ABB RAPID module: Module1.mod

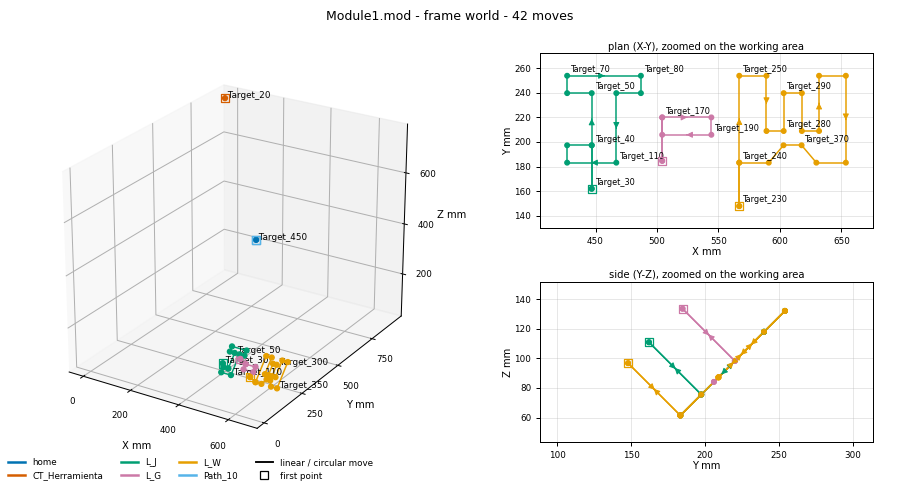
[picture p0: tool path of Module1.mod in frame world, 42 of 42 moves have a stored position in this frame; points joined in program order, loops and branches not executed]
MODULE Module1
    CONST robtarget Target_10:=[[-222.343363548,254.362,580.474563215],[0.5,-0.707106782,0.5,0],[0,-2,1,0],[9E+09,9E+09,9E+09,9E+09,9E+09,9E+09]];
    CONST robtarget Target_20:=[[-918.327354836,-454.935,-37.497165761],[0,0.923879533,0,-0.382683432],[0,0,0,0],[9E+09,9E+09,9E+09,9E+09,9E+09,9E+09]];
    CONST robtarget Target_30:=[[80.000242707,20.000268516,50.000191823],[0,0.707106778,0.707106785,0],[0,0,0,0],[9E+09,9E+09,9E+09,9E+09,9E+09,9E+09]];
    CONST robtarget Target_40:=[[80.000242721,20.000268516,0.000191823],[0,0.707106778,0.707106785,0],[0,0,0,0],[9E+09,9E+09,9E+09,9E+09,9E+09,9E+09]];
    CONST robtarget Target_50:=[[20.000242721,20.000268516,0.000191806],[0,0.707106778,0.707106785,0],[0,0,0,0],[9E+09,9E+09,9E+09,9E+09,9E+09,9E+09]];
    CONST robtarget Target_60:=[[20.000242721,0.000268516,0.000191806],[0,0.707106778,0.707106785,0],[0,0,0,0],[9E+09,9E+09,9E+09,9E+09,9E+09,9E+09]];
    CONST robtarget Target_70:=[[0.000242721,0.000268516,0.000191801],[0,0.707106778,0.707106785,0],[0,0,0,0],[9E+09,9E+09,9E+09,9E+09,9E+09,9E+09]];
    CONST robtarget Target_80:=[[0.000242721,60.000268516,0.000191801],[0,0.707106778,0.707106785,0],[0,0,0,0],[9E+09,9E+09,9E+09,9E+09,9E+09,9E+09]];
    CONST robtarget Target_90:=[[20.000242721,60.000268516,0.000191806],[0,0.707106778,0.707106785,0],[0,0,0,0],[9E+09,9E+09,9E+09,9E+09,9E+09,9E+09]];
    CONST robtarget Target_100:=[[20.000242721,40.000268516,0.000191806],[0,0.707106778,0.707106785,0],[0,0,0,0],[9E+09,9E+09,9E+09,9E+09,9E+09,9E+09]];
    CONST robtarget Target_110:=[[100.000242721,40.000268516,0.000191829],[0,0.707106778,0.707106785,0],[0,0,0,0],[9E+09,9E+09,9E+09,9E+09,9E+09,9E+09]];
    CONST robtarget Target_120:=[[100.000242721,0.000268516,0.000191829],[0,0.707106778,0.707106785,0],[0,0,0,0],[9E+09,9E+09,9E+09,9E+09,9E+09,9E+09]];
    CONST robtarget Target_130:=[[80.000242721,0.000268516,0.000191823],[0,0.707106778,0.707106785,0],[0,0,0,0],[9E+09,9E+09,9E+09,9E+09,9E+09,9E+09]];
    CONST robtarget Target_140:=[[80.000242721,20.000268516,0.000191823],[0,0.707106778,0.707106785,0],[0,0,0,0],[9E+09,9E+09,9E+09,9E+09,9E+09,9E+09]];
    CONST robtarget Target_150:=[[80.000242707,20.000268516,50.000191823],[0,0.707106778,0.707106785,0],[0,0,0,0],[9E+09,9E+09,9E+09,9E+09,9E+09,9E+09]];
    CONST robtarget Target_160:=[[47.906568131,77.338217332,50.000191814],[0,0.000000017,1,0],[0,0,0,0],[9E+09,9E+09,9E+09,9E+09,9E+09,9E+09]];
    CONST robtarget Target_170:=[[47.906568146,77.338217332,0.000191814],[0,0.000000017,1,0],[0,0,0,0],[9E+09,9E+09,9E+09,9E+09,9E+09,9E+09]];
    CONST robtarget Target_180:=[[47.906568146,117.338217332,0.000191814],[0,0.000000017,1,0],[0,0,0,0],[9E+09,9E+09,9E+09,9E+09,9E+09,9E+09]];
    CONST robtarget Target_190:=[[67.906568146,117.338217332,0.000191821],[0,0.000000017,1,0],[0,0,0,0],[9E+09,9E+09,9E+09,9E+09,9E+09,9E+09]];
    CONST robtarget Target_200:=[[67.906568146,77.338217332,0.000191821],[0,0.000000017,1,0],[0,0,0,0],[9E+09,9E+09,9E+09,9E+09,9E+09,9E+09]];
    CONST robtarget Target_210:=[[47.906568146,77.338217332,0.000191814],[0,0.000000017,1,0],[0,0,0,0],[9E+09,9E+09,9E+09,9E+09,9E+09,9E+09]];
    CONST robtarget Target_220:=[[47.906568131,77.338217332,50.000191814],[0,0.000000017,1,0],[0,0,0,0],[9E+09,9E+09,9E+09,9E+09,9E+09,9E+09]];
    CONST robtarget Target_230:=[[100.000242707,140.035099392,50.00019183],[0,-0.000000014,1,0],[0,0,0,0],[9E+09,9E+09,9E+09,9E+09,9E+09,9E+09]];
    CONST robtarget Target_240:=[[100.000242721,140.035099392,0.000191829],[0,-0.000000014,1,0],[0,0,0,0],[9E+09,9E+09,9E+09,9E+09,9E+09,9E+09]];
    CONST robtarget Target_250:=[[0.000242721,140.035099392,0.000191801],[0,-0.000000014,1,0],[0,0,0,0],[9E+09,9E+09,9E+09,9E+09,9E+09,9E+09]];
    CONST robtarget Target_260:=[[0.000242721,162.183714048,0.000191801],[0,-0.000000014,1,0],[0,0,0,0],[9E+09,9E+09,9E+09,9E+09,9E+09,9E+09]];
    CONST robtarget Target_270:=[[63.576949896,162.183714048,0.000191819],[0,-0.000000014,1,0],[0,0,0,0],[9E+09,9E+09,9E+09,9E+09,9E+09,9E+09]];
    CONST robtarget Target_280:=[[63.576949896,176.183714048,0.000191819],[0,-0.000000014,1,0],[0,0,0,0],[9E+09,9E+09,9E+09,9E+09,9E+09,9E+09]];
    CONST robtarget Target_290:=[[20.000242721,176.183714048,0.000191806],[0,-0.000000014,1,0],[0,0,0,0],[9E+09,9E+09,9E+09,9E+09,9E+09,9E+09]];
    CONST robtarget Target_300:=[[20.000242721,190.968722015,0.000191806],[0,-0.000000014,1,0],[0,0,0,0],[9E+09,9E+09,9E+09,9E+09,9E+09,9E+09]];
    CONST robtarget Target_310:=[[63.576949896,190.968722015,0.000191819],[0,-0.000000014,1,0],[0,0,0,0],[9E+09,9E+09,9E+09,9E+09,9E+09,9E+09]];
    CONST robtarget Target_320:=[[63.576949896,204.968722015,0.000191819],[0,-0.000000014,1,0],[0,0,0,0],[9E+09,9E+09,9E+09,9E+09,9E+09,9E+09]];
    CONST robtarget Target_330:=[[0.000242721,204.968722015,0.000191801],[0,-0.000000014,1,0],[0,0,0,0],[9E+09,9E+09,9E+09,9E+09,9E+09,9E+09]];
    CONST robtarget Target_340:=[[0.000242721,226.76231277,0.000191801],[0,-0.000000014,1,0],[0,0,0,0],[9E+09,9E+09,9E+09,9E+09,9E+09,9E+09]];
    CONST robtarget Target_350:=[[100.000242721,226.76231277,0.000191829],[0,-0.000000014,1,0],[0,0,0,0],[9E+09,9E+09,9E+09,9E+09,9E+09,9E+09]];
    CONST robtarget Target_360:=[[100.000242721,202.76231277,0.000191829],[0,-0.000000014,1,0],[0,0,0,0],[9E+09,9E+09,9E+09,9E+09,9E+09,9E+09]];
    CONST robtarget Target_370:=[[80.000242721,190.76231277,0.000191823],[0,-0.000000014,1,0],[0,0,0,0],[9E+09,9E+09,9E+09,9E+09,9E+09,9E+09]];
    CONST robtarget Target_380:=[[80.000242721,176.035099392,0.000191823],[0,-0.000000014,1,0],[0,0,0,0],[9E+09,9E+09,9E+09,9E+09,9E+09,9E+09]];
    CONST robtarget Target_390:=[[100.000242721,164.035099392,0.000191829],[0,-0.000000014,1,0],[0,0,0,0],[9E+09,9E+09,9E+09,9E+09,9E+09,9E+09]];
    CONST robtarget Target_400:=[[100.000242721,140.035099392,0.000191829],[0,-0.000000014,1,0],[0,0,0,0],[9E+09,9E+09,9E+09,9E+09,9E+09,9E+09]];
    CONST robtarget Target_410:=[[100.000242707,140.035099392,50.00019183],[0,-0.000000014,1,0],[0,0,0,0],[9E+09,9E+09,9E+09,9E+09,9E+09,9E+09]];
    CONST robtarget Target_450:=[[-216.657517919,253.804,577.362586272],[0.5,-0.707106781,0.5,0],[0,0,0,0],[9E+09,9E+09,9E+09,9E+09,9E+09,9E+09]];
    !***********************************************************
    !
    ! Módulo:  Module1
    !
    ! Descripción:
    !   <Introduzca la descripción aquí>
    !
    ! Autor: javie
    !
    ! Versión: 1.0
    !
    !***********************************************************


    !***********************************************************
    !
    ! Procedimiento Main
    !
    !   Este es el punto de entrada de su programa
    !
    !***********************************************************
    PROC main()
        !Añada aquí su código

        WaitDI EntDI_1,1;
        SetDO SalDO_1,1;
        CT_Herramienta;
        WaitDI EntDI_1,1;
        home;
        SetDO SalDO_1,0;

        WaitDI EntDI_2,1;
        SetDO SalDO_2,1;
        L_J;
        L_G;
        L_W;
        home;
        SetDO SalDO_2,0;
    ENDPROC

    PROC home()
        MoveJ Target_450,v100,z10,TCP_M\WObj:=WO_G03;
    ENDPROC
    PROC CT_Herramienta()
        MoveJ Target_20,v100,z10,TCP_M\WObj:=WO_G03;
    ENDPROC
    PROC L_J()
        MoveL Target_30,v100,z10,TCP_M\WObj:=WO_G03;
        MoveL Target_40,v100,z10,TCP_M\WObj:=WO_G03;
        MoveL Target_50,v100,z10,TCP_M\WObj:=WO_G03;
        MoveL Target_60,v100,z10,TCP_M\WObj:=WO_G03;
        MoveL Target_70,v100,z10,TCP_M\WObj:=WO_G03;
        MoveL Target_80,v100,z10,TCP_M\WObj:=WO_G03;
        MoveL Target_90,v100,z10,TCP_M\WObj:=WO_G03;
        MoveL Target_100,v100,z10,TCP_M\WObj:=WO_G03;
        MoveL Target_110,v100,z10,TCP_M\WObj:=WO_G03;
        MoveL Target_120,v100,z10,TCP_M\WObj:=WO_G03;
        MoveL Target_130,v100,z10,TCP_M\WObj:=WO_G03;
        MoveL Target_140,v100,z10,TCP_M\WObj:=WO_G03;
        MoveL Target_150,v100,z10,TCP_M\WObj:=WO_G03;
    ENDPROC
    PROC L_G()
        MoveL Target_160,v100,z10,TCP_M\WObj:=WO_G03;
        MoveL Target_170,v100,z10,TCP_M\WObj:=WO_G03;
        MoveL Target_180,v100,z10,TCP_M\WObj:=WO_G03;
        MoveL Target_190,v100,z10,TCP_M\WObj:=WO_G03;
        MoveL Target_200,v100,z10,TCP_M\WObj:=WO_G03;
        MoveL Target_210,v100,z10,TCP_M\WObj:=WO_G03;
        MoveL Target_220,v100,z10,TCP_M\WObj:=WO_G03;
    ENDPROC
    PROC L_W()
        MoveL Target_230,v100,z10,TCP_M\WObj:=WO_G03;
        MoveL Target_240,v100,z10,TCP_M\WObj:=WO_G03;
        MoveL Target_250,v100,z10,TCP_M\WObj:=WO_G03;
        MoveL Target_260,v100,z10,TCP_M\WObj:=WO_G03;
        MoveL Target_270,v100,z10,TCP_M\WObj:=WO_G03;
        MoveL Target_280,v100,z10,TCP_M\WObj:=WO_G03;
        MoveL Target_290,v100,z10,TCP_M\WObj:=WO_G03;
        MoveL Target_300,v100,z10,TCP_M\WObj:=WO_G03;
        MoveL Target_310,v100,z10,TCP_M\WObj:=WO_G03;
        MoveL Target_320,v100,z10,TCP_M\WObj:=WO_G03;
        MoveL Target_330,v100,z10,TCP_M\WObj:=WO_G03;
        MoveL Target_340,v100,z10,TCP_M\WObj:=WO_G03;
        MoveL Target_350,v100,z10,TCP_M\WObj:=WO_G03;
        MoveL Target_360,v100,z10,TCP_M\WObj:=WO_G03;
        MoveL Target_370,v100,z10,TCP_M\WObj:=WO_G03;
        MoveL Target_380,v100,z10,TCP_M\WObj:=WO_G03;
        MoveL Target_390,v100,z10,TCP_M\WObj:=WO_G03;
        MoveL Target_400,v100,z10,TCP_M\WObj:=WO_G03;
        MoveL Target_410,v100,z10,TCP_M\WObj:=WO_G03;
    ENDPROC
    PROC Path_10()
        MoveJ Target_450,v100,z10,TCP_M\WObj:=WO_G03;
    ENDPROC
ENDMODULE
